INTERFACE ITF_Cell

METHOD GetEmergencyOff : BOOL
VAR_INPUT
END_VAR
END_METHOD

METHOD GetEmergencyStop : BOOL
VAR_INPUT
END_VAR
END_METHOD

METHOD GetFinished : BOOL
VAR_INPUT
END_VAR
END_METHOD

METHOD GetIsRunning : BOOL
VAR_INPUT
END_VAR
END_METHOD

METHOD GetLoadPos : BOOL
VAR_INPUT
END_VAR
END_METHOD

METHOD GetStandby : BOOL
VAR_INPUT
END_VAR
END_METHOD

METHOD GetStartable : BOOL
VAR_INPUT
END_VAR
END_METHOD

METHOD GetUnloadPos : BOOL
VAR_INPUT
END_VAR
END_METHOD

METHOD SetEmergencyOff : BOOL
VAR_INPUT
	b :BOOL;
END_VAR
END_METHOD

METHOD SetEmergencyStop : BOOL
VAR_INPUT
	b :BOOL;
END_VAR
END_METHOD

METHOD SetMoveToLoad : BOOL
VAR_INPUT
	b :BOOL;
END_VAR
END_METHOD

METHOD SetMoveToUnload : BOOL
VAR_INPUT
	b :BOOL;
END_VAR
END_METHOD

METHOD SetStandby : BOOL
VAR_INPUT
	b :BOOL;
END_VAR
END_METHOD

METHOD SetStart : BOOL
VAR_INPUT
	b :BOOL;
END_VAR
END_METHOD

END_INTERFACE

(* stored: Version 1.1.0.1, ProductVersion 3.1.4024.0
   Itf ITF_Cell: Id {26b2a786-19bf-4b18-a47a-c2671c0ee775}
   Method GetEmergencyOff: Id {43aaa448-fd89-479e-96d2-c8fdef521945}
   Method GetEmergencyStop: Id {998f1cfa-1bb6-44da-beba-0310498112e3}
   Method GetFinished: Id {33137999-5e16-46a9-8760-9d98062065c2}
   Method GetIsRunning: Id {27010d55-e584-49eb-b39a-737ccf38e67d}
   Method GetLoadPos: Id {4456d7c7-b1e4-4418-b783-1997f2886cfc}
   Method GetStandby: Id {b77ffb79-5591-4c7e-aae7-9b37a011c2ea}
   Method GetStartable: Id {f13cd248-9c46-40a5-bc9a-470a1581974c}
   Method GetUnloadPos: Id {0a187401-a44d-471b-8112-663f8898c522}
   Method SetEmergencyOff: Id {27c8de1a-cba4-4b5c-b034-77cac3922498}
   Method SetEmergencyStop: Id {e152b9f9-767c-4979-b56a-99e34fdbf887}
   Method SetMoveToLoad: Id {167bf510-7f2d-4e27-98f4-1d0a22120b6d}
   Method SetMoveToUnload: Id {b7b14d61-9b88-4447-a2c2-ae951d8b3582}
   Method SetStandby: Id {d08c804a-6e63-4eb9-b70e-f83b87d3da75}
   Method SetStart: Id {9d86f309-b0fb-4954-9c10-45e24e1371e1} *)
